PROGRAM LOG_TIME_STAMP
VAR
END_VAR
VAR_INPUT
	LocalTime: FB_LocalSystemTime;
	Local_Date	: STRING;
	Local_Time	: STRING;
END_VAR



//================================ Function Block

LocalTime(
		sNetID:= , 
		bEnable:= TRUE , 
		dwCycle:= 1, 
		dwOpt:= , 
		tTimeout:= ,
		bValid=> , 
		systemTime=> , 
		tzID=> );

//================================ Footer System Time

IF NOT LocalTime.bValid THEN
	RETURN;
END_IF
		
Local_Date := CONCAT (WORD_TO_STRING(LocalTime.systemTime.wYear),' - ');
Local_Date := CONCAT (Local_Date, WORD_TO_STRING(LocalTime.systemTime.wMonth));
Local_Date := CONCAT (Local_Date, ' - ');
Local_Date := CONCAT (Local_Date, WORD_TO_STRING(LocalTime.systemTime.wDay));

Local_Time := CONCAT (WORD_TO_STRING(LocalTime.systemTime.wHour),' : ');
Local_Time := CONCAT (Local_Time, WORD_TO_STRING(LocalTime.systemTime.wMinute));
Local_Time := CONCAT (Local_Time, ' : ');
Local_Time := CONCAT (Local_Time, WORD_TO_STRING(LocalTime.systemTime.wSecond));

END_PROGRAM

(* stored: Version 1.1.0.1, ProductVersion 3.1.4024.12
   POU LOG_TIME_STAMP: Id {bb3c5f6f-245b-43ea-8105-1eeed363118f}, SpecialFunc None *)
